PROGRAM P_OEE_Raport
// Zmienne pomocnicze
VAR
    sCurrentDate        : STRING(10) := '';  // Przechowuje aktualną datę (np. "2023-10-25")
    bNewDay             : BOOL := FALSE;     // Flaga wskazująca, że rozpoczął się nowy dzień
    hFile               : UINT := 0;        // Uchwyt pliku
    sFilePath           : T_MaxString := ''; // Ścieżka do pliku
    nBytesToWrite       : UDINT := 0;        // Liczba bajtów do zapisania
    sLineToWrite             : T_MaxString := ''; // Bufor na dane do zapisania
    dtString            : STRING(20) := '';  // Czas zmiany w formacie tekstowym
    fbFileSeek          : FB_FileSeek;       // Blok do pozycjonowania wskaźnika pliku
    fbFileTell          : FB_FileTell;       // Blok do odczytu pozycji wskaźnika pliku
    fbFileGets          : FB_FileGets;       // Blok do odczytu linii z pliku
    bFileIsEmpty        : BOOL := FALSE;     // Flaga wskazująca, czy plik jest pusty
	RisingEdge			:R_trig;
	bSaveManuel			:BOOL;
	Step				:INT;
	bBusy 				:BOOL;
	bError				:BOOL;
	nErrId				:UDINT;
	nIndex				:INT;
	sFolderPath: STRING(255) := 'C:\OEE\';
	fbFileOpen: FB_FileOpen;
    fbFileWrite: FB_FileWrite;
    fbFileClose: FB_FileClose;
	b10step:BOOL;
	rtrig10MinsWork :r_trig;
	tonworkfor10min	:TON;
	AStBadPackageReasonText :ARRAY[0..63] OF S_Information_Text;
    i : INT;
    aIdToName: ARRAY[11..24] OF WSTRING := [
        "Wadliwa butelka lub proces przerwany:","Waga za mała:","Waga za duża:",
        "Brak odłożenia platynki:", "Platynka źle położona:", "Platynka nie zgrzana:",
        "Brak nas.(Słomka):", "Brak nasadki za zakręcarkami:","Brak nasadki przed zakręcarką:",
        "Nie zakręcono zakręcarką szczękową:", "Nasadka źle zakręcona:", "ROPP nie nałożony", 
		"ROPP nie zakręcony","ROPP brak za stacją"];
	bWork10min: BOOL;
	tontimerforevery10min :ton;
END_VAR

// Główna logika
IF Step=0 THEN
	bError:=FALSE;
END_IF
rtrig10MinsWork(CLK:=P_ADS_OEE.btonDelayAfterStart);
tonworkfor10min(in:=bWork10min, PT:=T#5M);
tontimerforevery10min(in:=NOT bWork10min AND P_ADS_OEE.btonDelayAfterStart, PT:=T#5M);
IF rtrig10MinsWork.Q  OR bSaveManuel OR tontimerforevery10min.q THEN
	bWork10min:=TRUE;
END_IF
IF tonworkfor10min.Q THEN
	bWork10min:=FALSE;
END_IF
RisingEdge(CLK := bSaveManuel OR tonworkfor10min.q OR P_ADS_OEE.bCycleReset OR P_ADS_OEE.btonConfectionEnding);

IF rtrig10MinsWork.Q  OR RisingEdge.q THEN 
	FOR i := 0 TO 63 DO
	    IF (P_ADS_OEE.AStBadPackageReason[i].udiID >= 11) AND (P_ADS_OEE.AStBadPackageReason[i].udiID <= 24) THEN
	        AStBadPackageReasonText[i].desc := aIdToName[P_ADS_OEE.AStBadPackageReason[i].udiID];
	    ELSE
	        AStBadPackageReasonText[i].desc := "";
	    END_IF;
	   
	    AStBadPackageReasonText[i].wsDescription := P_ADS_OEE.AStBadPackageReason[i].wsDescription;
	END_FOR;
END_IF

CASE Step OF
    0:
        // Sprawdź, czy zmienił się dzień
        IF LEFT(WSTRING_TO_STRING(P_time.s_time_mainscreen), 10) <> sCurrentDate THEN
            sCurrentDate := LEFT(WSTRING_TO_STRING(P_time.s_time_mainscreen), 10);  // Zaktualizuj datę
            bNewDay := TRUE;  // Ustaw flagę nowego dnia
        END_IF

        // Jeśli wystąpiło zdarzenie zapisu lub zmiany receptury
        IF RisingEdge.Q THEN
            bBusy := TRUE;
            bError := FALSE;
            nErrId := 0;
            nIndex := 0;

            // Utwórz ścieżkę do pliku na podstawie aktualnej daty
            sFilePath := CONCAT(sFolderPath, 'OEE_Raport_');
            sFilePath := CONCAT(sFilePath, sCurrentDate);
            sFilePath := CONCAT(sFilePath, '.csv');

            Step := 10;  // Przejdź do kroku otwarcia pliku
        END_IF

    10:
        // Otwórz plik
        IF bNewDay THEN
            // Jeśli nowy dzień, otwórz plik w trybie zapisu (tworzy nowy plik)
            fbFileOpen(
                sNetId := '', 
                sPathName := sFilePath, 
                nMode := FOPEN_MODEWRITE OR FOPEN_MODETEXT, 
                ePath := PATH_GENERIC, 
                bExecute := TRUE
            );
            b10step := TRUE;
        ELSE
            // Jeśli stary dzień, otwórz plik w trybie dopisywania
            fbFileOpen(
                sNetId := '', 
                sPathName := sFilePath, 
                nMode := FOPEN_MODEAPPEND OR FOPEN_MODETEXT, 
                ePath := PATH_GENERIC, 
                bExecute := TRUE
            );
            b10step := TRUE;
        END_IF
        Step := 20;

    20:
        // Czekaj na otwarcie pliku
        fbFileOpen(bExecute := FALSE);
        IF NOT fbFileOpen.bBusy THEN
            IF fbFileOpen.bError THEN
                nErrId := fbFileOpen.nErrId;
                bError := TRUE;
                Step := 500;  // Przejdź do kroku obsługi błędów
            ELSE
                hFile := fbFileOpen.hFile;
                Step := 30;  // Przejdź do kroku weryfikacji pliku
            END_IF
        END_IF

    30:
        // Sprawdź, czy plik jest pusty (tylko dla nowego dnia)
        IF bNewDay THEN
            fbFileTell(
                sNetId := '', 
                hFile := hFile, 
                bExecute := TRUE
            );
            Step := 35;
        ELSE
            Step := 40;  // Pomijaj weryfikację dla starego dnia
        END_IF

    35:
        // Czekaj na odczyt pozycji wskaźnika pliku
        fbFileTell(bExecute := FALSE);
        IF NOT fbFileTell.bBusy THEN
            IF fbFileTell.nSeekPos = 0 THEN
                bFileIsEmpty := TRUE;  // Plik jest pusty
            ELSE
                bFileIsEmpty := FALSE; // Plik nie jest pusty
            END_IF
            Step := 40;
        END_IF

    40:
        // Przygotuj dane do zapisu
        IF NOT fbFileTell.bBusy THEN
            sLineToWrite := CONCAT(WSTRING_TO_STRING(P_time.s_time_mainscreen), '|');
			sLineToWrite := CONCAT(sLineToWrite, WSTRING_TO_STRING(gvl_recipe.s_recipe_name));
            sLineToWrite := CONCAT(sLineToWrite, '|');
			sLineToWrite := CONCAT(sLineToWrite, INT_TO_STRING(REAL_TO_INT(P_ADS_OEE.uiCounterBadBottles)));
			sLineToWrite := CONCAT(sLineToWrite, '|');
            sLineToWrite := CONCAT(sLineToWrite, INT_TO_STRING(REAL_TO_INT(P_ADS_OEE.uiCounterGoodBottles)));
			sLineToWrite := CONCAT(sLineToWrite, '|');
			sLineToWrite := CONCAT(sLineToWrite, WSTRING_TO_STRING(AStBadPackageReasonText[0].desc));
            sLineToWrite := CONCAT(sLineToWrite, ':');
            sLineToWrite := CONCAT(sLineToWrite, WSTRING_TO_STRING(AStBadPackageReasonText[0].wsDescription));
			sLineToWrite := CONCAT(sLineToWrite, '|');			
            sLineToWrite := CONCAT(sLineToWrite, WSTRING_TO_STRING(AStBadPackageReasonText[1].desc));
            sLineToWrite := CONCAT(sLineToWrite, ':');
            sLineToWrite := CONCAT(sLineToWrite, WSTRING_TO_STRING(AStBadPackageReasonText[1].wsDescription));
			sLineToWrite := CONCAT(sLineToWrite, '|');
			sLineToWrite := CONCAT(sLineToWrite, WSTRING_TO_STRING(AStBadPackageReasonText[2].desc));
            sLineToWrite := CONCAT(sLineToWrite, ':');                                     
            sLineToWrite := CONCAT(sLineToWrite, WSTRING_TO_STRING(AStBadPackageReasonText[2].wsDescription));
			sLineToWrite := CONCAT(sLineToWrite, '|');
			sLineToWrite := CONCAT(sLineToWrite, WSTRING_TO_STRING(AStBadPackageReasonText[3].desc));
            sLineToWrite := CONCAT(sLineToWrite, ':');
            sLineToWrite := CONCAT(sLineToWrite, WSTRING_TO_STRING(AStBadPackageReasonText[3].wsDescription));
			sLineToWrite := CONCAT(sLineToWrite, '|');
			sLineToWrite := CONCAT(sLineToWrite, WSTRING_TO_STRING(AStBadPackageReasonText[4].desc));
            sLineToWrite := CONCAT(sLineToWrite, ':');
            sLineToWrite := CONCAT(sLineToWrite, WSTRING_TO_STRING(AStBadPackageReasonText[4].wsDescription));
			sLineToWrite := CONCAT(sLineToWrite, '|');
			sLineToWrite := CONCAT(sLineToWrite, WSTRING_TO_STRING(AStBadPackageReasonText[5].desc));
            sLineToWrite := CONCAT(sLineToWrite, ':');
            sLineToWrite := CONCAT(sLineToWrite, WSTRING_TO_STRING(AStBadPackageReasonText[5].wsDescription));
			sLineToWrite := CONCAT(sLineToWrite, '|');
			sLineToWrite := CONCAT(sLineToWrite, WSTRING_TO_STRING(AStBadPackageReasonText[6].desc));
            sLineToWrite := CONCAT(sLineToWrite, ':');
            sLineToWrite := CONCAT(sLineToWrite, WSTRING_TO_STRING(AStBadPackageReasonText[6].wsDescription));
			sLineToWrite := CONCAT(sLineToWrite, '|');
			sLineToWrite := CONCAT(sLineToWrite, WSTRING_TO_STRING(AStBadPackageReasonText[7].desc));
            sLineToWrite := CONCAT(sLineToWrite, ':');
            sLineToWrite := CONCAT(sLineToWrite, WSTRING_TO_STRING(AStBadPackageReasonText[7].wsDescription));
			sLineToWrite := CONCAT(sLineToWrite, '|');
			sLineToWrite := CONCAT(sLineToWrite, WSTRING_TO_STRING(AStBadPackageReasonText[8].desc));
            sLineToWrite := CONCAT(sLineToWrite, ':');
            sLineToWrite := CONCAT(sLineToWrite, WSTRING_TO_STRING(AStBadPackageReasonText[8].wsDescription));
			sLineToWrite := CONCAT(sLineToWrite, '|');
			sLineToWrite := CONCAT(sLineToWrite, WSTRING_TO_STRING(AStBadPackageReasonText[9].desc));
            sLineToWrite := CONCAT(sLineToWrite, ':');
            sLineToWrite := CONCAT(sLineToWrite, WSTRING_TO_STRING(AStBadPackageReasonText[9].wsDescription));
			sLineToWrite := CONCAT(sLineToWrite, '|');
			sLineToWrite := CONCAT(sLineToWrite, WSTRING_TO_STRING(AStBadPackageReasonText[10].desc));
            sLineToWrite := CONCAT(sLineToWrite, ':');
            sLineToWrite := CONCAT(sLineToWrite, WSTRING_TO_STRING(AStBadPackageReasonText[10].wsDescription));
			sLineToWrite := CONCAT(sLineToWrite, '|');
			sLineToWrite := CONCAT(sLineToWrite, WSTRING_TO_STRING(AStBadPackageReasonText[11].desc));
            sLineToWrite := CONCAT(sLineToWrite, ':');
            sLineToWrite := CONCAT(sLineToWrite, WSTRING_TO_STRING(AStBadPackageReasonText[11].wsDescription));
			sLineToWrite := CONCAT(sLineToWrite, '|');
			sLineToWrite := CONCAT(sLineToWrite, WSTRING_TO_STRING(AStBadPackageReasonText[12].desc));
            sLineToWrite := CONCAT(sLineToWrite, ':');
            sLineToWrite := CONCAT(sLineToWrite, WSTRING_TO_STRING(AStBadPackageReasonText[12].wsDescription));
			sLineToWrite := CONCAT(sLineToWrite, '|');
			sLineToWrite := CONCAT(sLineToWrite, WSTRING_TO_STRING(AStBadPackageReasonText[13].desc));
            sLineToWrite := CONCAT(sLineToWrite, ':');
            sLineToWrite := CONCAT(sLineToWrite, WSTRING_TO_STRING(AStBadPackageReasonText[13].wsDescription));
			sLineToWrite := CONCAT(sLineToWrite, '|');
			sLineToWrite := CONCAT(sLineToWrite, 'Czas pracy(min):');
			sLineToWrite := CONCAT(sLineToWrite, UINT_TO_STRING(P_ADS_OEE.udiCounterExecuteTime));
			sLineToWrite := CONCAT(sLineToWrite, '$N');

            nBytesToWrite := LEN(sLineToWrite);

            // Zapisz dane do pliku
            fbFileWrite(
                sNetId := '', 
                hFile := hFile, 
                pWriteBuff := ADR(sLineToWrite), 
                cbWriteLen := nBytesToWrite, 
                bExecute := TRUE
            );
            Step := 50;
        ELSE
            Step := 300;  // Przejdź do kroku zamknięcia pliku
        END_IF

    50:
        // Czekaj na zakończenie zapisu
        fbFileWrite(bExecute := FALSE);
        IF NOT fbFileWrite.bBusy THEN
            IF fbFileWrite.bError THEN
                nErrId := fbFileWrite.nErrId;
                bError := TRUE;
                Step := 500;  // Przejdź do kroku obsługi błędów
            ELSE
                Step := 300;  // Przejdź do kroku zamknięcia pliku po jednokrotnym zapisie
            END_IF
        END_IF

    300:
        // Zamknij plik
        fbFileClose(
            sNetId := '', 
            hFile := hFile, 
            bExecute := TRUE
        );
        Step := 310;

    310:
        // Czekaj na zamknięcie pliku
        fbFileClose(bExecute := FALSE);
        IF NOT fbFileClose.bBusy THEN
            IF fbFileClose.bError THEN
                nErrId := fbFileClose.nErrId;
                bError := TRUE;
            END_IF
            Step := 500;  // Przejdź do kroku obsługi błędów
        END_IF

    500:
        // Zakończ procedurę
        bBusy := FALSE;
        bNewDay := FALSE;  // Zresetuj flagę nowego dnia
        Step := 0;
END_CASE

END_PROGRAM

(* stored: Version 1.1.0.1, ProductVersion 3.1.4026.13, FileIdentifier c13cbad9e690958d135de3f6fc5cd260fa7b41c9, FileSignature 0a5b787a290aa329eab1b2e6077ecb2e88c5289a5439e291c1d11468424aa81adc68ced32554459be7592c86f9a0598e6eeb538e0cce9c012df92c33a67cc2dc77d1d2d9938f34f1b8f5d50b2d2469c336e81135fede2555ab277f8d0f5d0c8fa9fec312d9d7bd74b40bd1b91e71a5468933ff6859a8cbe637b03aba09db270208287d528874d22b4b8087c3122f6062419b53eade06819751b79fb0a2373a8bbe2afdb130210b2a972453344d70578306d79b3558600b3fb35a99c3c8a91b76806fb100e4757c03cd012d8638beb21748e565ce6d66039772a1b415520f50fb5ed7310d5b072b2418d155099aebe65ed352a6f474036ea2a2eea81b404e8fe6
   POU P_OEE_Raport: Id {fa602746-fe2d-4b96-9b8e-0aea45f807b4}, SpecialFunc None *)
